// TIA Portal V18 export
FUNCTION "fcFixtureCheck" : Void   // FC2, LAD
{ S7_Optimized_Access := 'TRUE' }
// stored: SetENOAutomatically false
   VAR_INPUT
      iRecipeSetValue : Byte;   // 配方设定工装值
   END_VAR
   VAR_IN_OUT
      FixtureIDCheck : Struct
         FixtureIDSetValue : Int;
         FixtureIDCheckValue : Int;
         FixtureCheckResult : Bool;
         FixtureCheckUnEnable : Bool;   // 工装检测使能,不需要检测时，给1
      END_STRUCT;
   END_VAR
BEGIN

REGION Network 2: 配方设定工装值 / Formula set tooling values
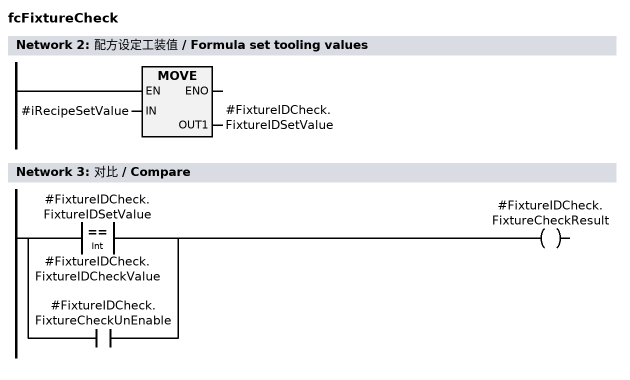
   RUNG wire#powerrail
      Move(in := #iRecipeSetValue, out1 => #FixtureIDCheck.FixtureIDSetValue)
   END_RUNG
   // the same network as SCL:
   #FixtureIDCheck.FixtureIDSetValue := #iRecipeSetValue;
END_REGION

REGION Network 3: 对比 / Compare
   RUNG wire#powerrail
      { S7_Templates := "SrcType := Int" } EQ_Contact(in1 := #FixtureIDCheck.FixtureIDSetValue, in2 := #FixtureIDCheck.FixtureIDCheckValue)
      wire#w1
      Coil( #FixtureIDCheck.FixtureCheckResult )
   END_RUNG
   RUNG wire#powerrail
      Contact( #FixtureIDCheck.FixtureCheckUnEnable )
   END_RUNG wire#w1
   // the same network as SCL:
   #FixtureIDCheck.FixtureCheckResult := (#FixtureIDCheck.FixtureIDSetValue = #FixtureIDCheck.FixtureIDCheckValue) OR #FixtureIDCheck.FixtureCheckUnEnable;
END_REGION
END_FUNCTION
